FUNCTION_BLOCK FB_LightControl_Dali implements I_LightControl
VAR_INPUT
END_VAR
VAR_OUTPUT
END_VAR
VAR
END_VAR

{warning 'add method implementation'}
METHOD M_Reset : BOOL
END_METHOD

{warning 'add method implementation'}
METHOD M_Set : BOOL
END_METHOD

{warning 'add property implementation'}
PROPERTY nAddress : DINT
GET
END_GET
SET
END_SET
END_PROPERTY

{warning 'add property implementation'}
PROPERTY nIlluminance : REAL
GET
END_GET
SET
END_SET
END_PROPERTY

END_FUNCTION_BLOCK

(* stored: Version 1.1.0.1, ProductVersion 3.1.4022.18
   POU FB_LightControl_Dali: Id {0e241490-0d03-4d44-820c-6de711c3af98}, SpecialFunc None
   Method M_Reset: Id {57d9b78d-f339-423f-804f-b3c5f5194cf9}
   Method M_Set: Id {a012e4cd-c6ff-416a-9f38-c0933b0a66ea}
   Property nAddress: Id {138c7b6f-ab66-4248-a0b5-771c08220421}
   Get Get: Id {dc42b859-0099-492a-9c10-cc25905fe907}
   Set Set: Id {7e4f999b-1b25-4ec3-8168-53ee78b8af33}
   Property nIlluminance: Id {93fa0e0f-14a1-41a5-8f5c-2cc45cd55bc7}
   Get Get: Id {fd4352fd-d141-4652-b6cf-2dd9341273ca}
   Set Set: Id {68c68892-dfd1-461a-99f3-41e1fa21c007} *)
